{attribute 'no_explicit_call' := 'direct call for this function block is not allowed'}
FUNCTION_BLOCK FINAL FB_EmptyWithRPC
VAR
END_VAR

// A method with all types of input and outputs as well as a return type.
{attribute 'TcRpcEnable'}
METHOD FullMethod : UDINT
VAR_INPUT
	InArg1  	: STRING(64);
	InArg2		: Tc2_System.ST_CpuCoreInfo; 
END_VAR
VAR_IN_OUT
	InOutArg1	: POINTER TO __UXINT;
END_VAR
VAR_OUTPUT
	OutArg1		: Tc2_System.E_SeekOrigin;
	OutArg2		: Tc2_System.T_MaxString;
END_VAR
END_METHOD

// First property.
{attribute 'TcRpcEnable'}
PROPERTY Prop1 : BOOL
GET
END_GET
SET
END_SET
END_PROPERTY

// A method that has no arguments.
{attribute 'TcRpcEnable'}
METHOD VoidMethod
VAR_INPUT
END_VAR
END_METHOD

END_FUNCTION_BLOCK

(* stored: Version 1.1.0.1, ProductVersion 3.1.4024.15
   POU FB_EmptyWithRPC: Id {349fa1b1-ed79-4982-b377-ab6a112fd293}, SpecialFunc None
   Method FullMethod: Id {5a84afde-7480-446d-ae1b-9735cdef484e}
   Property Prop1: Id {0c2e5a28-05c4-4305-916c-a535159ffd58}
   Get Get: Id {001ebcea-9997-4651-bd7c-552ca2559e74}
   Set Set: Id {e098534b-94f6-4880-a9d1-3d9d00e0c236}
   Method VoidMethod: Id {2ad03c31-41ce-466e-8158-002c54ce81d7} *)
